PROGRAM P200_CapPreScrewer
VAR_INPUT
	bEnable											: BOOL;	 										// Aktywacja bloku stacji					
	bRun											: BOOL; 
  	bPreRun											: BOOL; 
	bPlacePermission								: BOOL;                  				
	bHoming											: BOOL;                    				
	bManualMode										: BOOL;                     					// Tryb manualny
	bReset											: BOOL; 
	bIgnoreError									: BOOL;                    				
	iStationIndex									: UDINT		:= 1130;							// Numer stacji 
	wsStationName									: WSTRING	:= "Wkładacz zamknięć";		// Nazwa stacji
	stParameters									: ST_CapPreScrewerParameters := (	tTimeVacuumWatchdog		:= T#500MS,
																					lrTopZPosition				:= 400,
																					lrPickZPosition				:= 364,
																					lrPickYPosition				:= 26,
																					lrPlaceZPosition 			:= 236,		
																					lrCartesianCatchZPosition	:= 240,
																					lrPlaceYPosition 			:= 265,
																					lrCapCatcherZPosition 		:= 245,								
																					lrStrawCatcherZPosition 	:= 240,
																					LrCheckStrawCatcherActuatorZPosition:= 238,
																					lrScrewerStartZPosition 	:= 230,
																					lrCapCapCatcherRelese 		:= 228,
																					lrCatcherTopPosition 		:= 150,
																					lrCatcherCatchingPosition 	:= 130,
																					lrCatcherPlacePosition 		:= 70,
																					lrBendingDistance			:= 30,
																					lrScrewDistance				:= 180,
																					lrStrawInsertDistance 		:= 50,
																					lrCatcherSpeed 				:= 15,
																					lrPickerSpeed 				:= 15,
																					lrScrewSpeed 				:= 90,
																					lrCatcherMaxHight			:= 249,
																					lrCatcherMinHight			:= 0,
																					rCatcherHightOffset			:= 250,
																					lrCatcherHightSV			:= 90,	
																					rPulseRatio					:= 0.0140209058,
																					lrCatcherJerk				:= 100_000.0,
																					lrPickerJerk				:= 100_000.0,
																					lrScrewJerk					:= 1_000_000.0,
																					bRejectON					:= TRUE);
	
	
	//Wejścia sprzętowe
	bCapSuckerVacumOk1						: BOOL;		//Sygnał podciśnienia na ssawce nakrętki 1
	bCapSuckerVacumOk2						: BOOL;		//Sygnał podciśnienia na ssawce nakrętki 2
	bCapSuckerVacumOk3						: BOOL;		//Sygnał podciśnienia na ssawce nakrętki 3
	bCapSuckerVacumOk4						: BOOL;		//Sygnał podciśnienia na ssawce nakrętki 4
	
	diCapSuckerVacumOk1				AT%I*	: DINT;
    diCapSuckerVacumOk2				AT%I*	: DINT;
    diCapSuckerVacumOk3				AT%I*	: DINT;
    diCapSuckerVacumOk4				AT%I*	: DINT;

	iCapSuckerVacumOk1				AT%I*	: INT;
    iCapSuckerVacumOk2				AT%I*	: INT;
    iCapSuckerVacumOk3				AT%I*	: INT;
    iCapSuckerVacumOk4				AT%I*	: INT;
	
	
	bStrawCatcherOut		AT	%I*			: BOOL;		//Sygnał z krańcówki - wysunięty łapacz słomek
	bStrawCatcherIn			AT	%I*			: BOOL;		//Sygnał z krańcówki - wysunięty łapacz słomek
	
	bStrawCatcherOpen1		AT	%I*			: BOOL;		//Sygnał z krańcówki - otwart łapacz słomek 1
	bStrawCatcherOpen2		AT	%I*			: BOOL;		//Sygnał z krańcówki - otwart łapacz słomek 2
	bStrawCatcherOpen3		AT	%I*			: BOOL;		//Sygnał z krańcówki - otwart łapacz słomek 3
	bStrawCatcherOpen4		AT	%I*			: BOOL;		//Sygnał z krańcówki - otwart łapacz słomek 4
	
	bPendantDownwardMovement	AT%I*		: BOOL;			// Kaseta sterownicza ruch do góry
	bPendantUpwardMovement		AT%I*		: BOOL; 		// Kaseta sterownicza ruch do dolu
	bPendantUpDownFast			AT%I*		: BOOL;			// Kaseta sterownicza góra/dól- wyższa prędkośc
	bPendantRightwardMovement	AT%I*		: BOOL; 		// Kaseta sterownicza ruch w prawo
	bPendantLeftwardMovement	AT%I*		: BOOL; 		// Kaseta sterownicza ruch w lewo
	bPendantRightLeftFast		AT%I*		: BOOL;			// Kaseta sterownicza lewo/prawo- wyższa prędkośc
	
	bManualBottleGripperUp					: BOOL;
	bManualBottleGripperDown				: BOOL;
	
	bManualCartesianYJogPlus		: BOOL;			//Ruch ręczny podajnika zamknięć 
	bManualCartesianYJogMinus		: BOOL;			//Ruch ręczny podajnika zamknięć 
	bManualCartesianZJogPlus		: BOOL;			//Ruch ręczny podajnika zamknięć 
	bManualCartesianZJogMinus		: BOOL;			//Ruch ręczny podajnika zamknięć 
	
	bManualPreScrewerJogPlus		: BOOL;
	bManualPreScrewerJogMinus		: BOOL;
	
	bManualCatcherJogPlus			: BOOL;
	bManualCatcherJogMinus			: BOOL;
	bSimulationEna					: BOOL;
END_VAR

VAR_OUTPUT
	bBottleGrippers				AT	%Q*		: BOOL;						//Sygnał do zaworu - łapania szyjek butelek

	bCapSucker1					AT	%Q*		: BOOL;						//Sygnał do zaworu - zassij nakrętkę 1
	bCapSucker2					AT	%Q*		: BOOL;						//Sygnał do zaworu - zassij nakrętkę 2
	bCapSucker3					AT	%Q*		: BOOL;						//Sygnał do zaworu - zassij nakrętkę 3
	bCapSucker4					AT	%Q*		: BOOL;						//Sygnał do zaworu - zassij nakrętkę 4
	
	bCapBlower1					AT	%Q*		: BOOL;						//Sygnał do zaworu - wydmuchaj nakrętkę 1
	bCapBlower2					AT	%Q*		: BOOL;						//Sygnał do zaworu - wydmuchaj nakrętkę 2
	bCapBlower3					AT	%Q*		: BOOL;						//Sygnał do zaworu - wydmuchaj nakrętkę 3
	bCapBlower4					AT	%Q*		: BOOL;						//Sygnał do zaworu - wydmuchaj nakrętkę 4
	
	bCapCatcher1				AT	%Q*		: BOOL;						//Sygnał do zaworu - złap nakrętkę 1
	bCapCatcher2				AT	%Q*		: BOOL;						//Sygnał do zaworu - złap nakrętkę 2
	bCapCatcher3				AT	%Q*		: BOOL;						//Sygnał do zaworu - złap nakrętkę 3
	bCapCatcher4				AT	%Q*		: BOOL;						//Sygnał do zaworu - złap nakrętkę 4
	
	bStrawCatchersOpen			AT	%Q*		: BOOL;						//Sygnał do zaworu - otwórz chwytaki słomek
	bStrawCatchersClose			AT	%Q*		: BOOL;						//Sygnał do zaworu - zamknij chwytaki słomek
	
	bStrawCatcherActuatorOut	AT	%Q*		: BOOL;						//Sygnał do zaworu - wysuń łapacz słomek
	bStrawCatcherActuatorIn		AT	%Q*		: BOOL;						//Sygnał do zaworu - wsuń łapacz słomek
	
	
	eState									: E_Station;								// Stan ogólny bloku
	eRunnigState							: E_CapPreScrewer;
	bError									: BOOL;										// Błąd bloku
	udiErrorID								: UDINT;									// Numer błędu
	sErrorDescription1						: STRING(200);								// Opis błędu 1
	sErrorDescription2						: STRING(200);								// Opis błędu 2
	sErrorStationName						: STRING;									// Nazwa stacji
	bHomingDone								: BOOL;										// Stacja zbazowana
	bCycleNotDone							: BOOL;										// Cykl nie został wykonany
	bCycleDone								: BOOL;										// Cykl został wykonany
	aCapPresence							: ARRAY [1..4] OF BOOL;
	bAnyCapSucker							: BOOL;										//Przynajmniej jedna nakrętka pobrana
	bRejectDone								: BOOL;
END_VAR



VAR
	fbCapPreScrewer							: FB_CapPreScrewer;
	fbCapPreScrewerState					: FB_State;
	
	bTestRun								: BOOL;
	bTestHoming								: BOOL;
	bTestReset								: BOOL;
	
	tonCheckVacuum							: TON;
	tCycleTime								: TIME;
	bMissingCaps							: BOOL;

	bCartesianSafePos						: BOOL;
	stCommandsIN							: ST_CapPreScrewerCommandsIn;
	bTestEnable: BOOL;
	bCapSuckerTemp: ARRAY [1..4] OF  BOOL;
	bVacuumTest: BOOL;
	bTestPreRun: BOOL;
	tonCapCatcher1	: TON;
	tonCapCatcher2	: TON;
	tonCapCatcher3	: TON;
	tonCapCatcher4	: TON;
	fbVacuumInputFilter	: ARRAY [1..4] OF FB_FilterEx;
	bTestSettingStation	: BOOL;
	ftTestSettingStation	: F_TRIG;
	fbTimeFilter	: FB_DigitalInput_1;
END_VAR



IF bCapSucker4 AND NOT bCapSuckerVacumOk4 AND eState = E_Station.eRunning  THEN
	tCycleTime			:= tonCheckVacuum.ET;
END_IF

tonCheckVacuum(IN := bCapSucker4 AND NOT bCapSuckerVacumOk4, PT := T#2D);

GVL_VIS.bCapSorterPreScrewerCatcherStationHeightSet := SEL((ABS(GVL_VIS.lrCapSorterPreScrewerCatcherStationHeightCV-GVL_Recipe.lrCapSorterPreScrewerCatcherHightSVShow)<=1.0),
													GVL_VIS.bCapSorterPreScrewerCatcherStationHeightSet, FALSE);

//*****************Sterowanie zaworami ssawek***********************************
bCapSucker1 := NOT stparameters.bvacuumDeactivate AND bCapSuckerTemp[1];
bCapSucker2 := NOT stparameters.bvacuumDeactivate AND bCapSuckerTemp[2];
bCapSucker3 := NOT stparameters.bvacuumDeactivate AND bCapSuckerTemp[3];
bCapSucker4 := NOT stparameters.bvacuumDeactivate AND bCapSuckerTemp[4];

stParameters.LrCheckStrawCatcherActuatorZPosition;
stParameters.lrStrawCatcherZPosition;
stParameters.lrCartesianCatchZPosition;

//bAnyCapSucker := bCapSucker1 OR bCapSucker2 OR bCapSucker3 OR bCapSucker4;
//fbCapPreScrewer.stMoverStatus := SEL(P190_CapFeeder.stMover1Status.bInPlacePosition, P190_CapFeeder.stMover2Status, P190_CapFeeder.stMover1Status);

//_____________________Generowanie stanu do wizki______________________________________
fbCapPreScrewerState(	eState 					:= eState,
			 			bRun					:= bRun,
			 			sStateDesc				=> GVL_VIS.sCapSorterPreScrewerState,
			 			iState					=> GVL_VIS.iCapSorterPreScrewerState);
				
stParameters.lrPickerSpeedWhenScrewer;

ACT_FB();

//Adresy dla komunikacji ADS
stParameters.sADS_NetId					:= '192.168.40.160.4.1';
stParameters.nAxisY_ADS_SlaveAddr		:= 1020;
stParameters.nAxisZ_ADS_SlaveAddr		:= 1020;
stParameters.nCatcher_ADS_SlaveAddr		:= 1019;


//Przepisanie zmiennych
stCommandsIN.bPendantDownwardMovement	:= bPendantDownwardMovement	;
stCommandsIN.bPendantUpwardMovement		:= bPendantUpwardMovement	;	
stCommandsIN.bPendantUpDownFast			:= bPendantUpDownFast		;	
stCommandsIN.bPendantRightwardMovement	:= bPendantRightwardMovement;	
stCommandsIN.bPendantLeftwardMovement	:= bPendantLeftwardMovement	;
stCommandsIN.bPendantRightLeftFast		:= bPendantRightLeftFast	;	
//stCommandsIN.bChoseRecipe				:= GVL_Communication.bChooseRecipe;


GVL_Recipe.lrCapSorterPreScrewerPickXMover1PositionShow			;
GVL_recipe.lrCapSorterPreScrewerPlaceXPositionShow			;
GVL_recipe.lrCapSorterPreScrewerTopZPositionShow			;
GVL_recipe.lrCapSorterPreScrewerPickZPositionShow			;
GVL_recipe.lrCapSorterPreScrewerCatcherCatchingPositionShow	;
GVL_recipe.lrCapSorterPreScrewerCartesianCatchZPositionShow;
GVL_recipe.LrCapSorterPreScrewerCheckStrawCatcherActuatorZPosition;
GVL_recipe.lrCapSorterPreScrewerPlaceZPositionShow			;
GVL_recipe.lrCapSorterPreScrewerCapCatcherZPositionShow		;
GVL_recipe.lrCapSorterPreScrewerGripperOpenPositionShow		;
GVL_recipe.lrCapSorterPreScrewerCatcherReleseShow			;
GVL_recipe.lrCapSorterPreScrewerStrawCatcherZPositionShow	;
GVL_recipe.lrCapSorterPreScrewerScrewerStartZPositionShow	;
GVL_recipe.lrCapSorterPreScrewerBendingDistanceShow			;
                                                            
GVL_Recipe.lrCapSorterPreScrewerCatcherHightSVShow			;
GVL_Recipe.lrCapSorterPreScrewerCatcherCatchingPositionShow	;
GVL_Recipe.lrCapSorterPreScrewerCatcherPlacePositionShow	;
                                                            
GVL_recipe.lrCapSorterPreScrewerScrewDistanceShow			;
GVL_recipe.lrCapSorterPreScrewerStrawInsertDistance			;
                                                            
GVL_Recipe.lrCapSorterPreScrewerCatcherSpeedShow			;
GVL_Recipe.lrCapSorterPreScrewerPickerSpeedShow				;
GVL_Recipe.lrCapSorterPreScrewerScrewSpeedShow				;
                                                            
GVL_Recipe.lrCapSorterPreScrewerCatcherHightSVShow			;


stParameters.bPickerActiv[1];

stParameters.rCatcherHightOffset ;

// bCapSuckerVacumOk1			:= ABS(diCapSuckerVacumOk1) >= 450;	
// bCapSuckerVacumOk2			:= ABS(diCapSuckerVacumOk2) >= 450;	
// bCapSuckerVacumOk3			:= ABS(diCapSuckerVacumOk3) >= 450;	
// bCapSuckerVacumOk4			:= ABS(diCapSuckerVacumOk4) >= 450;	
fbVacuumInputFilter[1](rIn := INT_TO_REAL(iCapSuckerVacumOk1), tTimeConstant	:= T#25MS);
fbVacuumInputFilter[2](rIn := INT_TO_REAL(iCapSuckerVacumOk2), tTimeConstant	:= T#25MS);
fbVacuumInputFilter[3](rIn := INT_TO_REAL(iCapSuckerVacumOk3), tTimeConstant	:= T#25MS);
fbVacuumInputFilter[4](rIn := INT_TO_REAL(iCapSuckerVacumOk4), tTimeConstant	:= T#25MS);


GVL_VIS.lrCapSorterPreScrewerVacuumLevel_1	:= DINT_TO_LREAL(iCapSuckerVacumOk1)/10_000;
GVL_VIS.lrCapSorterPreScrewerVacuumLevel_2	:= DINT_TO_LREAL(iCapSuckerVacumOk2)/10_000;
GVL_VIS.lrCapSorterPreScrewerVacuumLevel_3	:= DINT_TO_LREAL(iCapSuckerVacumOk3)/10_000;
GVL_VIS.lrCapSorterPreScrewerVacuumLevel_4	:= DINT_TO_LREAL(iCapSuckerVacumOk4)/10_000;

bCapSuckerVacumOk1			:= ABS(iCapSuckerVacumOk1/10) >= 480;	
bCapSuckerVacumOk2			:= ABS(iCapSuckerVacumOk2/10) >= 480;	
bCapSuckerVacumOk3			:= ABS(iCapSuckerVacumOk3/10) >= 480;	
bCapSuckerVacumOk4			:= ABS(iCapSuckerVacumOk4/10) >= 480;	

tonCapCatcher1(IN := bCapCatcher1, PT := T#100MS);
tonCapCatcher2(IN := bCapCatcher2, PT := T#100MS);
tonCapCatcher3(IN := bCapCatcher3, PT := T#100MS);
tonCapCatcher4(IN := bCapCatcher4, PT := T#100MS);




IF bTestSettingStation THEN
	IF GVL_VIS.lrCapSorterPreScrewerCatcherStationHeightCV < 300 AND NOT GVL_VIS.bCapSorterPreScrewerCatcherStationDown THEN
		fbTimeFilter.In	:= TRUE;
		GVL_VIS.bCapSorterPreScrewerCatcherStationUp	:= fbTimeFilter.bIn;
	ELSIF GVL_VIS.lrCapSorterPreScrewerCatcherStationHeightCV >= 300 THEN
		fbTimeFilter.In	:= FALSE;
		GVL_VIS.bCapSorterPreScrewerCatcherStationUp	:= FALSE;
		GVL_VIS.bCapSorterPreScrewerCatcherStationDown 	S= NOT fbTimeFilter.bIn;
	ELSIF GVL_VIS.lrCapSorterPreScrewerCatcherStationHeightCV <= 100 THEN
		GVL_VIS.bCapSorterPreScrewerCatcherStationDown 	:= FALSE;	
	END_IF	
ELSIF ftTestSettingStation.Q THEN
	fbTimeFilter.In	:= FALSE;
	GVL_VIS.bCapSorterPreScrewerCatcherStationUp	:= FALSE;
	GVL_VIS.bCapSorterPreScrewerCatcherStationDown 	:= FALSE;		
END_IF

fbTimeFilter.tTimeOn 	:= T#500MS;
fbTimeFilter.tTimeOff	:= T#500mS;
fbTimeFilter.FilterTrig();
ftTestSettingStation(CLK := bTestSettingStation);

ACTION ACT_FB:
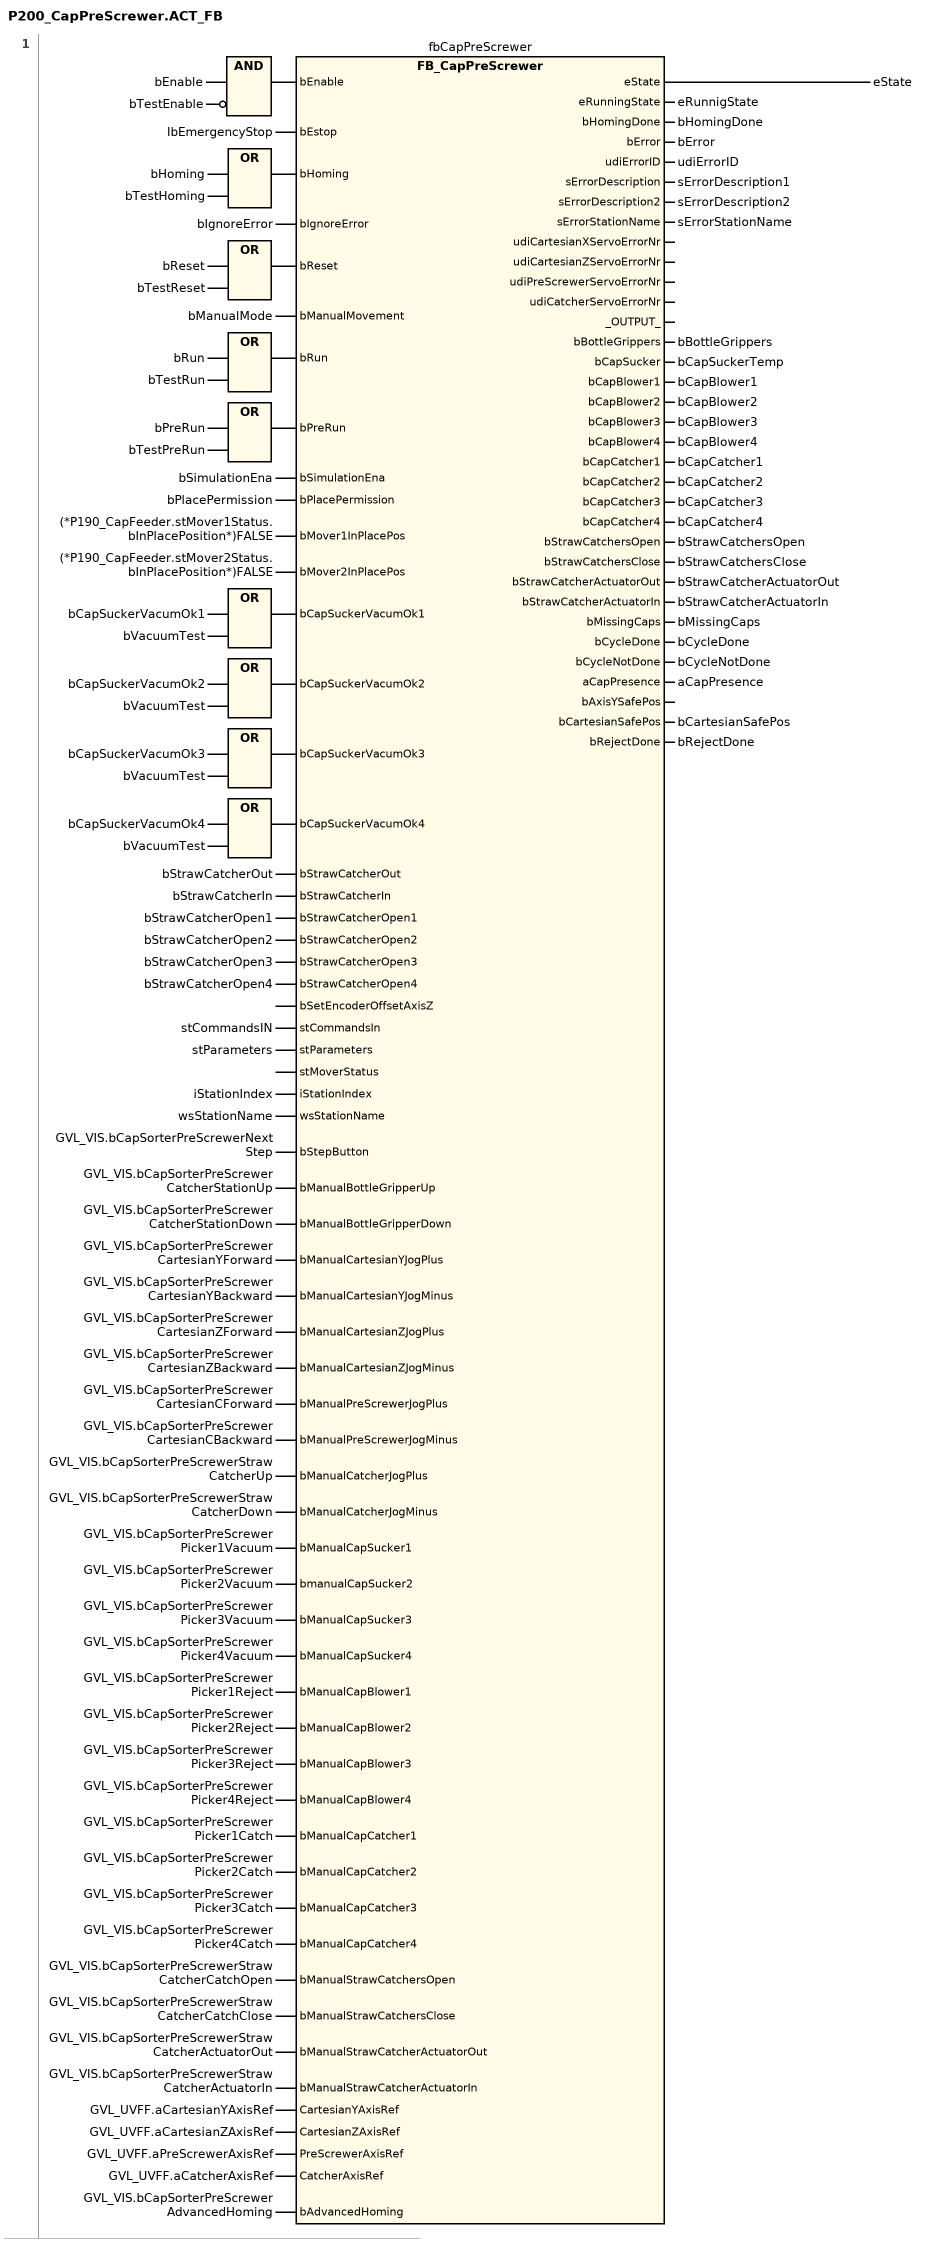
// NETWORK 1
fbCapPreScrewer(
    bEnable := bEnable AND NOT bTestEnable,
    bEstop := IbEmergencyStop,
    bHoming := bHoming OR bTestHoming,
    bIgnoreError := bIgnoreError,
    bReset := bReset OR bTestReset,
    bManualMovement := bManualMode,
    bRun := bRun OR bTestRun,
    bPreRun := bPreRun OR bTestPreRun,
    bSimulationEna := bSimulationEna,
    bPlacePermission := bPlacePermission,
    bMover1InPlacePos := (*P190_CapFeeder.stMover1Status.bInPlacePosition*)FALSE,
    bMover2InPlacePos := (*P190_CapFeeder.stMover2Status.bInPlacePosition*)FALSE,
    bCapSuckerVacumOk1 := bCapSuckerVacumOk1 OR bVacuumTest,
    bCapSuckerVacumOk2 := bCapSuckerVacumOk2 OR bVacuumTest,
    bCapSuckerVacumOk3 := bCapSuckerVacumOk3 OR bVacuumTest,
    bCapSuckerVacumOk4 := bCapSuckerVacumOk4 OR bVacuumTest,
    bStrawCatcherOut := bStrawCatcherOut,
    bStrawCatcherIn := bStrawCatcherIn,
    bStrawCatcherOpen1 := bStrawCatcherOpen1,
    bStrawCatcherOpen2 := bStrawCatcherOpen2,
    bStrawCatcherOpen3 := bStrawCatcherOpen3,
    bStrawCatcherOpen4 := bStrawCatcherOpen4,
    stCommandsIn := stCommandsIN,
    stParameters := stParameters,
    iStationIndex := iStationIndex,
    wsStationName := wsStationName,
    bStepButton := GVL_VIS.bCapSorterPreScrewerNextStep,
    bManualBottleGripperUp := GVL_VIS.bCapSorterPreScrewerCatcherStationUp,
    bManualBottleGripperDown := GVL_VIS.bCapSorterPreScrewerCatcherStationDown,
    bManualCartesianYJogPlus := GVL_VIS.bCapSorterPreScrewerCartesianYForward,
    bManualCartesianYJogMinus := GVL_VIS.bCapSorterPreScrewerCartesianYBackward,
    bManualCartesianZJogPlus := GVL_VIS.bCapSorterPreScrewerCartesianZForward,
    bManualCartesianZJogMinus := GVL_VIS.bCapSorterPreScrewerCartesianZBackward,
    bManualPreScrewerJogPlus := GVL_VIS.bCapSorterPreScrewerCartesianCForward,
    bManualPreScrewerJogMinus := GVL_VIS.bCapSorterPreScrewerCartesianCBackward,
    bManualCatcherJogPlus := GVL_VIS.bCapSorterPreScrewerStrawCatcherUp,
    bManualCatcherJogMinus := GVL_VIS.bCapSorterPreScrewerStrawCatcherDown,
    bManualCapSucker1 := GVL_VIS.bCapSorterPreScrewerPicker1Vacuum,
    bmanualCapSucker2 := GVL_VIS.bCapSorterPreScrewerPicker2Vacuum,
    bManualCapSucker3 := GVL_VIS.bCapSorterPreScrewerPicker3Vacuum,
    bManualCapSucker4 := GVL_VIS.bCapSorterPreScrewerPicker4Vacuum,
    bManualCapBlower1 := GVL_VIS.bCapSorterPreScrewerPicker1Reject,
    bManualCapBlower2 := GVL_VIS.bCapSorterPreScrewerPicker2Reject,
    bManualCapBlower3 := GVL_VIS.bCapSorterPreScrewerPicker3Reject,
    bManualCapBlower4 := GVL_VIS.bCapSorterPreScrewerPicker4Reject,
    bManualCapCatcher1 := GVL_VIS.bCapSorterPreScrewerPicker1Catch,
    bManualCapCatcher2 := GVL_VIS.bCapSorterPreScrewerPicker2Catch,
    bManualCapCatcher3 := GVL_VIS.bCapSorterPreScrewerPicker3Catch,
    bManualCapCatcher4 := GVL_VIS.bCapSorterPreScrewerPicker4Catch,
    bManualStrawCatchersOpen := GVL_VIS.bCapSorterPreScrewerStrawCatcherCatchOpen,
    bManualStrawCatchersClose := GVL_VIS.bCapSorterPreScrewerStrawCatcherCatchClose,
    bManualStrawCatcherActuatorOut := GVL_VIS.bCapSorterPreScrewerStrawCatcherActuatorOut,
    bManualStrawCatcherActuatorIn := GVL_VIS.bCapSorterPreScrewerStrawCatcherActuatorIn,
    CartesianYAxisRef := GVL_UVFF.aCartesianYAxisRef,
    CartesianZAxisRef := GVL_UVFF.aCartesianZAxisRef,
    PreScrewerAxisRef := GVL_UVFF.aPreScrewerAxisRef,
    CatcherAxisRef := GVL_UVFF.aCatcherAxisRef,
    bAdvancedHoming := GVL_VIS.bCapSorterPreScrewerAdvancedHoming,
    eRunningState => eRunnigState,
    bHomingDone => bHomingDone,
    bError => bError,
    udiErrorID => udiErrorID,
    sErrorDescription => sErrorDescription1,
    sErrorDescription2 => sErrorDescription2,
    sErrorStationName => sErrorStationName,
    bBottleGrippers => bBottleGrippers,
    bCapSucker => bCapSuckerTemp,
    bCapBlower1 => bCapBlower1,
    bCapBlower2 => bCapBlower2,
    bCapBlower3 => bCapBlower3,
    bCapBlower4 => bCapBlower4,
    bCapCatcher1 => bCapCatcher1,
    bCapCatcher2 => bCapCatcher2,
    bCapCatcher3 => bCapCatcher3,
    bCapCatcher4 => bCapCatcher4,
    bStrawCatchersOpen => bStrawCatchersOpen,
    bStrawCatchersClose => bStrawCatchersClose,
    bStrawCatcherActuatorOut => bStrawCatcherActuatorOut,
    bStrawCatcherActuatorIn => bStrawCatcherActuatorIn,
    bMissingCaps => bMissingCaps,
    bCycleDone => bCycleDone,
    bCycleNotDone => bCycleNotDone,
    aCapPresence => aCapPresence,
    bCartesianSafePos => bCartesianSafePos,
    bRejectDone => bRejectDone); // FB_CapPreScrewer
eState := fbCapPreScrewer.eState;
END_ACTION

END_PROGRAM

(* stored: Version 1.2.0.0, ProductVersion 3.1.4026.13, FileIdentifier f46dbf2eb7b3b1ebf424352a3445bcd578b76ec7, FileSignature 0f6f019dbe176d1c082754c84fbd826b8f5d09d0a77aa5d4a6cffa1c553fa6c75a81a709a2093069bea5ead58e3428215f6f961121f44ce7205be3e011dc28960d8bff2bb54fde0f6b1978fc914cceca03419a4b047ac8950e538ca7d8c73dfe12ff78eb0b6f4d3381d6c48009d43a141f7eaee36ac7c7c1f84f53d2945da9230da494b196127029993cf12661cfb00ff245d1b6e2efd3da3d6a7d1fecba77d9a3f06b295d90355218ee4b44fba1354d5b1a4820335c765ee369eb8a1562eb7c17b96c5f0ea6e2f2f13e7acc32c68653e52e6bc653428308c78b8e6f6ec007fc328b76c747bb55faa22c6013564b4b4dc71198c64affdcd75cc848cd6e09f5a1
   POU P200_CapPreScrewer: Id {27d184ef-d145-4fcb-8ac2-b1a7f6a870b2}, SpecialFunc None
   Action ACT_FB: Id {9339763c-40f9-4dc4-9cf9-92aaf7c3c8c1} *)
